KUKA KRL program: wkz1_an.src, wkz1_an.dat

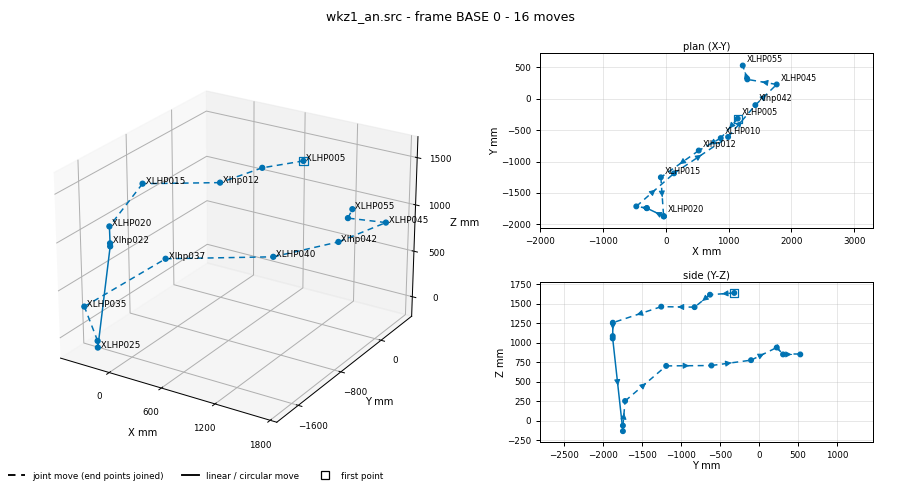
[picture p0: tool path of wkz1_an.src in frame BASE 0, 16 of 16 moves have a stored position in this frame; points joined in program order, loops and branches not executed]
--- wkz1_an.src ---
&ACCESS RVP4
&REL 450
&COMMENT Retira pinca C1
&PARAM DISKPATH = KRC:\R1\Program
DEF wkz1_an( )
;FOLD INI
   ;FOLD BASISTECH INI
      GLOBAL INTERRUPT DECL 3 WHEN $STOPMESS==TRUE DO IR_STOPM ( )
      INTERRUPT ON 3
      BAS (#INITMOV,0 )
   ;ENDFOLD (BASISTECH INI)
   ;FOLD SPOTTECH INI
      USERSPOT(#INIT)
   ;ENDFOLD (SPOTTECH INI)
   ;FOLD GRIPPERTECH INI
      USER_GRP(0,DUMMY,DUMMY,GDEFAULT)
   ;ENDFOLD (GRIPPERTECH INI)
   ;FOLD USER INI
      ;Make your modifications here

   ;ENDFOLD (USER INI)
;ENDFOLD (INI)

; Estacao P13.060 - Robo R1
; Programa: Busca Pinça C1
; Info: Gun F2 6640 0018 991
; Caracterização dos meios de produção:
; 02/09/2014 09:15 Changes by KUKA Roboter do Brasil

chk_w8_wechs_ok ( )   ; CHECK FERRAMENTA: TOOL CHANGE

;FOLD OUT 168 'DOCK1 Fechar Protecao' State=FALSE CONT;%{PE}%R 8.2.20,%MKUKATPBASIS,%COUT,%VOUTX,%P 2:168, 3:DOCK1 Fechar Protecao, 5:FALSE, 6:CONTINUE
CONTINUE
$OUT[168]=FALSE
;ENDFOLD
;FOLD PULSE 167 'DOCK1 Abrir Protecao' State=TRUE CONT Time=3 sec;%{PE}%R 8.2.20,%MKUKATPBASIS,%COUT,%VPULSE,%P 2:167, 3:DOCK1 Abrir Protecao, 5:TRUE, 6:CONTINUE, 8:3
CONTINUE
PULSE($OUT[167], TRUE,3)
;ENDFOLD

;FOLD PTP LHP005 Vel=80 % PDAT12 Tool[8]:Tool Changer Base[0];%{PE}%R 8.2.20,%MKUKATPBASIS,%CMOVE,%VPTP,%P 1:PTP, 2:LHP005, 3:, 5:80, 7:PDAT12
$BWDSTART=FALSE
PDAT_ACT=PPDAT12
FDAT_ACT=FLHP005
BAS(#PTP_PARAMS,80)
PTP XLHP005
;ENDFOLD

;FOLD WAIT FOR IN 161 'deposito ocupado'  State= TRUE ;%{PE}%R 4.1.16,%MKUKATPBASIS,%CWAIT_FOR,%VWAIT_FOR,%P 1:0, 2:161, 3:'deposito ocupado', 5:TRUE, 6:
WAIT FOR $IN[161]==TRUE
;ENDFOLD
;FOLD WAIT FOR IN 219 'placas de suporte fundidas'  State= FALSE ;%{PE}%R 4.1.16,%MKUKATPBASIS,%CWAIT_FOR,%VWAIT_FOR,%P 1:0, 2:219, 3:'placas de suporte fundidas', 5:FALSE, 6:
WAIT FOR $IN[219]==FALSE
;ENDFOLD
;FOLD WAIT FOR IN 165 'protecao da pinca aberto'  State= TRUE ;%{PE}%R 4.1.16,%MKUKATPBASIS,%CWAIT_FOR,%VWAIT_FOR,%P 1:0, 2:165, 3:'protecao da pinca aberto', 5:TRUE, 6:
WAIT FOR $IN[165]==TRUE
;ENDFOLD

;FOLD PTP LHP010 CONT Vel= 100 % P_OLP2 Tool[1]:GUN C1 Base[0];%{PE}%R 4.1.16,%MKUKATPBASIS,%CMOVE,%VPTP,%P 1:PTP, 2:LHP010, 3:C_PTP, 5:100, 7:P_OLP2
$BWDSTART = FALSE
PDAT_ACT=PP_OLP2
BAS(#PTP_DAT)
FDAT_ACT=FLHP010
BAS(#FRAMES)
BAS(#VEL_PTP,100)
PTP XLHP010 C_PTP
;ENDFOLD
;FOLD PTP lhp012 CONT Vel=90 % PDAT5 Tool[1]:GUN C1 Base[0];%{PE}%R 8.2.20,%MKUKATPBASIS,%CMOVE,%VPTP,%P 1:PTP, 2:lhp012, 3:C_DIS, 5:90, 7:PDAT5
$BWDSTART=FALSE
PDAT_ACT=PPDAT5
FDAT_ACT=Flhp012
BAS(#PTP_PARAMS,90)
PTP Xlhp012 C_DIS
;ENDFOLD

;FOLD PTP LHP015 CONT Vel=90 % PDAT1 Tool[1]:GUN C1 Base[0];%{PE}%R 8.2.20,%MKUKATPBASIS,%CMOVE,%VPTP,%P 1:PTP, 2:LHP015, 3:C_DIS, 5:90, 7:PDAT1
$BWDSTART=FALSE
PDAT_ACT=PPDAT1
FDAT_ACT=FLHP015
BAS(#PTP_PARAMS,90)
PTP XLHP015 C_DIS
;ENDFOLD
;FOLD PTP LHP020 Vel=70 % PDAT3 Tool[8]:Tool Changer Base[0];%{PE}%R 8.2.20,%MKUKATPBASIS,%CMOVE,%VPTP,%P 1:PTP, 2:LHP020, 3:, 5:70, 7:PDAT3
$BWDSTART=FALSE
PDAT_ACT=PPDAT3
FDAT_ACT=FLHP020
BAS(#PTP_PARAMS,70)
PTP XLHP020
;ENDFOLD
;FOLD LIN lhp022 Vel=0.4 m/s CPDAT5 Tool[8]:Tool Changer Base[0];%{PE}%R 8.2.20,%MKUKATPBASIS,%CMOVE,%VLIN,%P 1:LIN, 2:lhp022, 3:, 5:0.4, 7:CPDAT5
$BWDSTART=FALSE
LDAT_ACT=LCPDAT5
FDAT_ACT=Flhp022
BAS(#CP_PARAMS,0.4)
LIN Xlhp022
;ENDFOLD

;FOLD WAIT FOR IN 222 'Klaschka ativado'  State= TRUE ;%{PE}%R 4.1.16,%MKUKATPBASIS,%CWAIT_FOR,%VWAIT_FOR,%P 1:0, 2:222, 3:'Klaschka ativado', 5:TRUE, 6:
WAIT FOR $IN[222]==TRUE
;ENDFOLD
;FOLD OUT 224 'Bloqueio MPS'  State= FALSE ;%{PE}%R 4.1.16,%MKUKATPBASIS,%COUT,%VOUTX,%P 2:224, 3:'Bloqueio MPS', 5:FALSE, 6:
$OUT[224]=FALSE
;ENDFOLD
;FOLD OUT 223 'Desbloqueio MPS'  State= TRUE ;%{PE}%R 4.1.16,%MKUKATPBASIS,%COUT,%VOUTX,%P 2:223, 3:'Desbloqueio MPS', 5:TRUE, 6:
$OUT[223]=TRUE
;ENDFOLD
;FOLD WAIT FOR IN 217 'MPS destravado'  State= TRUE ;%{PE}%R 4.1.16,%MKUKATPBASIS,%CWAIT_FOR,%VWAIT_FOR,%P 1:0, 2:217, 3:'MPS destravado', 5:TRUE, 6:
WAIT FOR $IN[217]==TRUE
;ENDFOLD
;FOLD WAIT FOR IN 221 'MPS travado'  State= FALSE ;%{PE}%R 4.1.16,%MKUKATPBASIS,%CWAIT_FOR,%VWAIT_FOR,%P 1:0, 2:221, 3:'MPS travado', 5:FALSE, 6:
WAIT FOR $IN[221]==FALSE
;ENDFOLD

;FOLD ; PONTO_DE PEGA DA PINCA;%{PE}%R 4.1.16,%MKUKATPBASIS,%CCOMMENT,%VNORMAL,%P 2:PONTO_DE PEGA DA PINCA
;ENDFOLD
;FOLD LIN PickPos_Gun01  Vel=2.0 m/s CPDAT3 Tool[8] Base[0];%{PE}%R 4.1.15,%MKUKATPBASIS,%CMOVE,%VLIN,%P 1:LIN, 2:PickPos_Gun01, 3:, 5:2.0, 7:CPDAT3
$BWDSTART=FALSE
LDAT_ACT=LCPDAT3
BAS(#CP_DAT )
FDAT_ACT=FPickPos_Gun01
BAS(#FRAMES )
BAS(#VEL_CP,2.0 )
LIN  XPickPos_Gun01
;ENDFOLD

;FOLD WAIT FOR IN 219 'placas de suporte fundidas'  State= TRUE ;%{PE}%R 4.1.16,%MKUKATPBASIS,%CWAIT_FOR,%VWAIT_FOR,%P 1:0, 2:219, 3:'placas de suporte fundidas', 5:TRUE, 6:
WAIT FOR $IN[219]==TRUE
;ENDFOLD
;FOLD IBUS  OFF;%{PE}%R 4.1.16,%MKUKATPBASIS,%CIBUS,%VMAP,%P 2:#OFF, 3:1
$IBUS_OFF=$IBUS_ON
$IBUS_ON=0
;ENDFOLD
;FOLD OUT 223 'Desbloqueio MPS'  State= FALSE ;%{PE}%R 4.1.16,%MKUKATPBASIS,%COUT,%VOUTX,%P 2:223, 3:'Desbloqueio MPS', 5:FALSE, 6:
$OUT[223]=FALSE
;ENDFOLD
;FOLD OUT 224 'Bloqueio MPS'  State= TRUE ;%{PE}%R 4.1.16,%MKUKATPBASIS,%COUT,%VOUTX,%P 2:224, 3:'Bloqueio MPS', 5:TRUE, 6:
$OUT[224]=TRUE
;ENDFOLD
;FOLD WAIT FOR IN 221 'MPS travado'  State= TRUE ;%{PE}%R 4.1.16,%MKUKATPBASIS,%CWAIT_FOR,%VWAIT_FOR,%P 1:0, 2:221, 3:'MPS travado', 5:TRUE, 6:
WAIT FOR $IN[221]==TRUE
;ENDFOLD
;FOLD WAIT FOR IN 217 'MPS destravado'  State= FALSE ;%{PE}%R 4.1.16,%MKUKATPBASIS,%CWAIT_FOR,%VWAIT_FOR,%P 1:0, 2:217, 3:'MPS destravado', 5:FALSE, 6:
WAIT FOR $IN[217]==FALSE
;ENDFOLD
;FOLD WAIT 0.5 0 sec;%{PE}%R 8.2.20,%MKUKATPBASIS,%CWAIT,%VWAIT,%P 3:0
WAIT SEC 0
;ENDFOLD
;FOLD IBUS  ON SEGMENT_1;%{PE}%R 4.1.16,%MKUKATPBASIS,%CIBUS,%VMAP,%P 2:#ON, 3:1
$IBUS_ON=IBUS_SEGMENT[1]
$IBUS_OFF=0
;ENDFOLD
;FOLD ; INICIO DA SAIDA COM A PINCA;%{PE}%R 4.1.16,%MKUKATPBASIS,%CCOMMENT,%VNORMAL,%P 2:INICIO DA SAIDA COM A PINCA
;ENDFOLD
;FOLD LIN LHP025 CONT Vel=0.4 m/s CPDAT4 Tool[1]:GUN C1 Base[0];%{PE}%R 8.2.20,%MKUKATPBASIS,%CMOVE,%VLIN,%P 1:LIN, 2:LHP025, 3:C_DIS C_DIS, 5:0.4, 7:CPDAT4
$BWDSTART=FALSE
LDAT_ACT=LCPDAT4
FDAT_ACT=FLHP025
BAS(#CP_PARAMS,0.4)
LIN XLHP025 C_DIS C_DIS
;ENDFOLD
;FOLD LIN LHP030 CONT Vel= 0.6 m/s L_OLP1 Tool[1]:GUN C1 Base[0];%{PE}%R 4.1.16,%MKUKATPBASIS,%CMOVE,%VLIN,%P 1:LIN, 2:LHP030, 3:C_DIS, 5:0.6, 7:L_OLP1
$BWDSTART = FALSE
LDAT_ACT=LL_OLP1
BAS(#CP_DAT)
FDAT_ACT=FLHP030
BAS(#FRAMES)
BAS(#VEL_CP,0.6)
LIN XLHP030 C_DIS
;ENDFOLD

;FOLD WAIT FOR IN 161 'dock 1 ocupado'  State= FALSE ;%{PE}%R 4.1.16,%MKUKATPBASIS,%CWAIT_FOR,%VWAIT_FOR,%P 1:0, 2:161, 3:'dock 1 ocupado', 5:FALSE, 6:
WAIT FOR $IN[161]==FALSE
;ENDFOLD
;FOLD WAIT FOR IN 219 'placas de suporte fundidas'  State= TRUE ;%{PE}%R 4.1.16,%MKUKATPBASIS,%CWAIT_FOR,%VWAIT_FOR,%P 1:0, 2:219, 3:'placas de suporte fundidas', 5:TRUE, 6:
WAIT FOR $IN[219]==TRUE
;ENDFOLD

;FOLD PTP LHP035 CONT Vel=80 % PDAT4 Tool[1]:GUN C1 Base[0];%{PE}%R 8.2.20,%MKUKATPBASIS,%CMOVE,%VPTP,%P 1:PTP, 2:LHP035, 3:C_DIS, 5:80, 7:PDAT4
$BWDSTART=FALSE
PDAT_ACT=PPDAT4
FDAT_ACT=FLHP035
BAS(#PTP_PARAMS,80)
PTP XLHP035 C_DIS
;ENDFOLD
;FOLD PTP lhp037 CONT Vel=80 % PDAT6 Tool[1]:GUN C1 Base[0];%{PE}%R 8.2.20,%MKUKATPBASIS,%CMOVE,%VPTP,%P 1:PTP, 2:lhp037, 3:C_DIS, 5:80, 7:PDAT6
$BWDSTART=FALSE
PDAT_ACT=PPDAT6
FDAT_ACT=Flhp037
BAS(#PTP_PARAMS,80)
PTP Xlhp037 C_DIS
;ENDFOLD

;FOLD PTP LHP040 CONT Vel=80 % P_OLP5 Tool[1]:GUN C1 Base[0];%{PE}%R 8.2.20,%MKUKATPBASIS,%CMOVE,%VPTP,%P 1:PTP, 2:LHP040, 3:C_DIS, 5:80, 7:P_OLP5
$BWDSTART=FALSE
PDAT_ACT=PP_OLP5
FDAT_ACT=FLHP040
BAS(#PTP_PARAMS,80)
PTP XLHP040 C_DIS
;ENDFOLD
;FOLD PTP lhp042 CONT Vel=80 % PDAT8 Tool[1]:GUN C1 Base[0];%{PE}%R 8.2.20,%MKUKATPBASIS,%CMOVE,%VPTP,%P 1:PTP, 2:lhp042, 3:C_DIS, 5:80, 7:PDAT8
$BWDSTART=FALSE
PDAT_ACT=PPDAT8
FDAT_ACT=Flhp042
BAS(#PTP_PARAMS,80)
PTP Xlhp042 C_DIS
;ENDFOLD
;FOLD PTP LHP045 CONT Vel=80 % P_OLP6 Tool[1]:GUN C1 Base[0];%{PE}%R 8.2.20,%MKUKATPBASIS,%CMOVE,%VPTP,%P 1:PTP, 2:LHP045, 3:C_DIS, 5:80, 7:P_OLP6
$BWDSTART=FALSE
PDAT_ACT=PP_OLP6
FDAT_ACT=FLHP045
BAS(#PTP_PARAMS,80)
PTP XLHP045 C_DIS
;ENDFOLD
;FOLD PTP LHP050 CONT Vel=80 % PDAT7 Tool[1]:GUN C1 Base[0];%{PE}%R 8.2.20,%MKUKATPBASIS,%CMOVE,%VPTP,%P 1:PTP, 2:LHP050, 3:C_DIS, 5:80, 7:PDAT7
$BWDSTART=FALSE
PDAT_ACT=PPDAT7
FDAT_ACT=FLHP050
BAS(#PTP_PARAMS,80)
PTP XLHP050 C_DIS
;ENDFOLD
;FOLD PTP LHP055 CONT Vel=80 % PDAT2 Tool[1]:GUN C1 Base[0];%{PE}%R 8.2.20,%MKUKATPBASIS,%CMOVE,%VPTP,%P 1:PTP, 2:LHP055, 3:C_DIS, 5:80, 7:PDAT2
$BWDSTART=FALSE
PDAT_ACT=PPDAT2
FDAT_ACT=FLHP055
BAS(#PTP_PARAMS,80)
PTP XLHP055 C_DIS
;ENDFOLD


END

--- wkz1_an.dat ---
&ACCESS RVP4
&REL 450
&COMMENT Retira pinca C1
&PARAM DISKPATH = KRC:\R1\Program
DEFDAT  wkz1_an
;FOLD EXTERNAL DECLARATIONS;%{PE}%MKUKATPBASIS,%CEXT,%VCOMMON,%P
;FOLD GRIPPERTECH EXT
EXT  H50 (INT  :IN,INT  :IN,INT  :IN,GRP_TYP  :IN )
;ENDFOLD (GRIPPERTECH EXT)
;FOLD SPOTTECH EXT
EXT  USERSPOT (S_COMMAND  :IN,SPOT_TYPE  :IN )
;ENDFOLD (SPOTTECH EXT)
;FOLD BASISTECH EXT;%{PE}%MKUKATPBASIS,%CEXT,%VEXT,%P
EXT  BAS (BAS_COMMAND  :IN,REAL  :IN )
DECL INT SUCCESS
;ENDFOLD (BASISTECH EXT)
;FOLD USER EXT;%{E}%MKUKATPUSER,%CEXT,%VEXT,%P
;Make your modifications here

;ENDFOLD (USER EXT)
;ENDFOLD (EXTERNAL DECLARATIONS)

;# ============ START PATH : za_p13060r1_c1 =============
DECL FDAT FLHP010={TOOL_NO 8,BASE_NO 0,IPO_FRAME #BASE}
DECL PDAT PP_OLP2={VEL 100.0,ACC 75.0,APO_DIST 80.0}
DECL E6POS XLHP010={X 874.56958,Y -626.810974,Z 1613.96899,A -30.9093094,B -16.7809505,C 178.532898,S 18,T 2,E1 0.0,E2 0.0,E3 0.0,E4 0.0,E5 0.0,E6 0.0}
DECL FDAT FLHP015={TOOL_NO 8,BASE_NO 0,IPO_FRAME #BASE,TQ_STATE FALSE}
DECL E6POS XLHP015={X -79.4015884,Y -1250.95801,Z 1460.75696,A -16.15312,B -0.262848496,C -179.600494,S 18,T 10,E1 0.0,E2 0.0,E3 0.0,E4 0.0,E5 0.0,E6 0.0}
DECL FDAT FLHP020={TOOL_NO 8,BASE_NO 0,IPO_FRAME #BASE,TQ_STATE FALSE}
DECL E6POS XLHP020={X -35.1820297,Y -1871.13306,Z 1255.47302,A -10.6039305,B -0.565146327,C 179.772598,S 18,T 10,E1 0.0,E2 0.0,E3 0.0,E4 0.0,E5 0.0,E6 0.0}
DECL FDAT FLHP030={TOOL_NO 1,BASE_NO 0,IPO_FRAME #BASE}
DECL E6POS XLHP030={X -303.188507,Y -1742.18701,Z -62.3764801,A 154.739807,B 1.49047899,C -0.0905354023,S 18,T 10,E1 0.0,E2 0.0,E3 0.0,E4 0.0,E5 0.0,E6 0.0}
DECL LDAT LL_OLP1={VEL 0.25,ACC 75.0,APO_DIST 5.0,APO_FAC 0.0}
DECL FDAT FLHP035={TOOL_NO 1,BASE_NO 0,IPO_FRAME #BASE,TQ_STATE FALSE}
DECL E6POS XLHP035={X -470.50351,Y -1714.19397,Z 252.719604,A 159.801498,B 2.5038259,C 3.27011991,S 18,T 10,E1 0.0,E2 0.0,E3 0.0,E4 0.0,E5 0.0,E6 0.0}
DECL LDAT LL_OLP2={VEL 0.25,ACC 85.0,APO_DIST 50.0,APO_FAC 0.0}
DECL FDAT FLHP040={TOOL_NO 1,BASE_NO 0,IPO_FRAME #BASE}
DECL PDAT PP_OLP5={VEL 100.0,ACC 80.0,APO_DIST 30.0,APO_MODE #CDIS}
DECL E6POS XLHP040={X 992.169678,Y -608.116272,Z 706.993713,A -124.100304,B 6.65894699,C 18.2110901,S 18,T 10,E1 0.0,E2 0.0,E3 0.0,E4 0.0,E5 0.0,E6 0.0}
DECL FDAT FLHP045={TOOL_NO 1,BASE_NO 0,IPO_FRAME #BASE}
DECL PDAT PP_OLP6={VEL 100.0,ACC 75.0,APO_DIST 50.0,APO_MODE #CDIS}
DECL E6POS XLHP045={X 1765.87903,Y 228.156494,Z 937.730286,A 86.3647537,B -5.19986391,C -28.1547108,S 2,T 10,E1 0.0,E2 0.0,E3 0.0,E4 0.0,E5 0.0,E6 0.0}
DECL LDAT LCPDAT1={VEL 2.0,ACC 75.0,APO_DIST 20.0,APO_FAC 50.0}
DECL LDAT LCPDAT2={VEL 2.0,ACC 85.0,APO_DIST 3.0,APO_FAC 50.0}
DECL LDAT LCPDAT3={VEL 2.0,ACC 100.0,APO_DIST 100.0,APO_FAC 50.0}
DECL E6POS XLHP055={X 1225.07996,Y 529.6521,Z 849.202881,A 96.890358,B -6.64530277,C -11.59793,S 2,T 10,E1 0.0,E2 0.0,E3 0.0,E4 0.0,E5 0.0,E6 0.0}
DECL FDAT FLHP055={TOOL_NO 1,BASE_NO 0,IPO_FRAME #BASE}
DECL PDAT PPDAT2={VEL 100.0,ACC 75.0,APO_DIST 70.0,APO_MODE #CDIS}
DECL E6POS XLHP025={X -303.101501,Y -1742.12,Z -134.100693,A 154.739899,B 1.49296296,C -0.0887258276,S 18,T 10,E1 0.0,E2 0.0,E3 0.0,E4 0.0,E5 0.0,E6 0.0}
DECL FDAT FLHP025={TOOL_NO 1,BASE_NO 0,IPO_FRAME #BASE,TQ_STATE FALSE}
DECL LDAT LCPDAT4={VEL 2.0,ACC 85.0,APO_DIST 3.0,APO_FAC 50.0}
DECL E6POS XLHP050={X 1298.44299,Y 308.865601,Z 849.20282,A 86.8900681,B -6.64529085,C -11.59793,S 2,T 10,E1 0.0,E2 0.0,E3 0.0,E4 0.0,E5 0.0,E6 0.0}
DECL FDAT FLHP050={TOOL_NO 1,BASE_NO 0,IPO_FRAME #BASE}
DECL PDAT PPDAT7={VEL 100.0,ACC 75.0,APO_DIST 70.0,APO_MODE #CDIS}
DECL PDAT PPDAT12={VEL 80.0,ACC 100.0,APO_DIST 10.0}
DECL SPOT_SUGG_T LAST_SPOT={GUN[] "1                       ",RETR_CMD[] "#CLO                    ",CHOISE[] "#FIRST                  ",CLO_TM[] "1                       ",PGNO1[] "251                     ",PRESS1[] "0                       ",PGNO2[] "1                       ",PRESS2[] "0                       ",SPOT_PARAMS[] "NORMAL                  "}
DECL E6POS XLHP005={X 1144.98206,Y -315.997406,Z 1636.51794,A -70.0583496,B -10.0851498,C -166.622803,S 18,T 2,E1 0.0,E2 0.0,E3 0.0,E4 0.0,E5 0.0,E6 0.0}
DECL FDAT FLHP005={TOOL_NO 8,BASE_NO 0,IPO_FRAME #BASE,TQ_STATE FALSE}
DECL E6POS XPickPos_Gun01={X -30.9670792,Y -1872.86694,Z 1053.36597,A -10.2532701,B -1.18632698,C 179.471497,S 18,T 10,E1 0.0,E2 0.0,E3 0.0,E4 0.0,E5 0.0,E6 0.0}
DECL FDAT FPickPos_Gun01={TOOL_NO 8,BASE_NO 0,IPO_FRAME #BASE}
DECL BASIS_SUGG_T LAST_BASIS={POINT1[] "lhp042                  ",POINT2[] "lhp042                  ",CP_PARAMS[] "CPDAT5                  ",PTP_PARAMS[] "PDAT8                   ",CONT[] "C_DIS                   ",CP_VEL[] "0.4                     ",PTP_VEL[] "90                      ",SYNC_PARAMS[] "SYNCDAT                 ",SPL_NAME[] "S0                      "}
DECL PDAT PPDAT1={VEL 100.0,ACC 80.0,APO_DIST 80.0,APO_MODE #CDIS,GEAR_JERK 50.0}
DECL PDAT PPDAT3={VEL 100.0,ACC 80.0,APO_DIST 40.0,APO_MODE #CDIS,GEAR_JERK 50.0}
DECL E6POS XLHP022={X -31.5506992,Y -1872.47498,Z 1083.98096,A -10.2532196,B -1.18534994,C 179.472504,S 18,T 10,E1 0.0,E2 0.0,E3 0.0,E4 0.0,E5 0.0,E6 0.0}
DECL FDAT Flhp022={TOOL_NO 8,BASE_NO 0,IPO_FRAME #BASE,POINT2[] " ",TQ_STATE FALSE}
DECL LDAT LCPDAT5={VEL 2.0,ACC 85.0,APO_DIST 100.0,APO_FAC 50.0,AXIS_VEL 100.0,AXIS_ACC 100.0,ORI_TYP #VAR,CIRC_TYP #BASE,JERK_FAC 50.0,GEAR_JERK 50.0,EXAX_IGN 0}
DECL PDAT PPDAT4={VEL 100.0,ACC 80.0,APO_DIST 60.0,APO_MODE #CDIS,GEAR_JERK 50.0}
DECL E6POS XLHP007={X 524.31488,Y -824.293701,Z 1454.45703,A 18.5507202,B -1.67638099,C 174.630997,S 18,T 10,E1 0.0,E2 0.0,E3 0.0,E4 0.0,E5 0.0,E6 0.0}
DECL FDAT Flhp007={TOOL_NO 8,BASE_NO 0,IPO_FRAME #BASE,POINT2[] " ",TQ_STATE FALSE}
DECL PDAT PPDAT5={VEL 100.0,ACC 80.0,APO_DIST 25.0,APO_MODE #CDIS,GEAR_JERK 50.0}
DECL E6POS Xlhp012={X 524.31488,Y -824.293701,Z 1454.45703,A 18.5507202,B -1.67638099,C 174.630997,S 18,T 10,E1 0.0,E2 0.0,E3 0.0,E4 0.0,E5 0.0,E6 0.0}
DECL FDAT Flhp012={TOOL_NO 8,BASE_NO 0,IPO_FRAME #BASE,POINT2[] " ",TQ_STATE FALSE}
DECL E6POS XLHP037={X 130.042801,Y -1187.81299,Z 702.066284,A -178.5298,B 6.79400206,C 17.9013996,S 18,T 10,E1 0.0,E2 0.0,E3 0.0,E4 0.0,E5 0.0,E6 0.0}
DECL FDAT Flhp037={TOOL_NO 1,BASE_NO 0,IPO_FRAME #BASE,POINT2[] " ",TQ_STATE FALSE}
DECL PDAT PPDAT6={VEL 100.0,ACC 80.0,APO_DIST 50.0,APO_MODE #CDIS,GEAR_JERK 50.0}
DECL E6POS XLHP042={X 1425.63,Y -101.145401,Z 775.48407,A 125.505096,B 22.0524597,C -19.6151104,S 18,T 10,E1 0.0,E2 0.0,E3 0.0,E4 0.0,E5 0.0,E6 0.0}
DECL FDAT Flhp042={TOOL_NO 1,BASE_NO 0,IPO_FRAME #BASE,POINT2[] " ",TQ_STATE FALSE}
DECL PDAT PPDAT8={VEL 100.0,ACC 80.0,APO_DIST 30.0,APO_MODE #CDIS,GEAR_JERK 50.0}
ENDDAT
